PROGRAM main
  VAR
    BUTTON AT %QX0.0 : BOOL;
    MOTOR AT %QX0.1 : BOOL;
  END_VAR

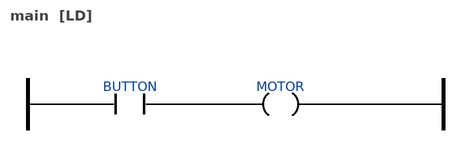
(* LD diagram, written out as Structured Text *)
MOTOR := BUTTON;
END_PROGRAM
